RoboDK station: PaintingUV.rdk

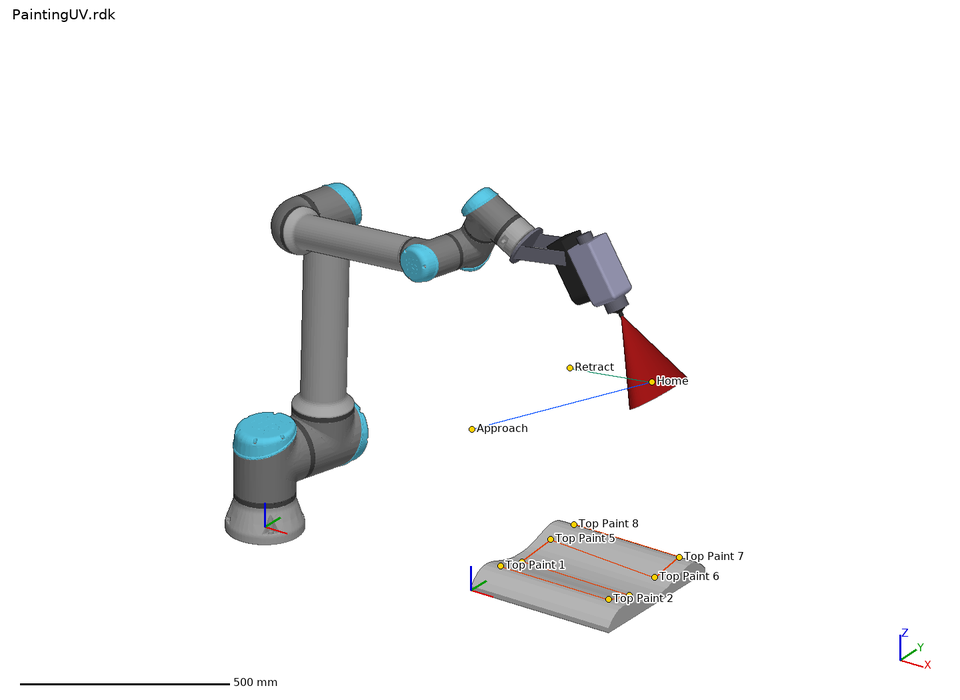
[picture v0: the station drawn from its stored meshes, robots at their saved joint values, targets as dots, program paths as lines]
Station PaintingUV (saved by RoboDK 5.9.0). Poses are relative to the parent item; angles as X-Y-Z fixed-axis rotations.
Station parameters (name, value as stored): LIN64
  - frame UR10e Base at (0, 0, 0) mm
    - robot UR10e: 6 axes, payload 10 kg, reach 1300 mm, repeatability 0.05 mm, weight 28.9 kg
        modified DH rows (alpha deg, a mm, theta deg, d mm): 0, 0, 0, 180.7; 90, 0, 180, 0; 0, 612.6, 0, 0; 0, 571.335, 0, 174.15; -90, 0, 0, 119.85; 90, 0, 180, 116.55
        joint limits [-360, -360, -360, -360, -360, -360] to [360, 360, 360, 360, 360, 360]; home [0, -90, -90, 0, 90, 0]; saved at [164.043, -88.205, 75.684, -137.69, -76.063, 82.15]
      - tool Paint gun, TCP at (50, 0, 450) mm, rotated rx 0 ry 30 rz 0 deg, size 203.2 x 279.7 x 471.5 mm
  - frame Frame 2 at (600, 0, 0) mm
    - object Object Inspection at (0, 0, 0) mm, size 400 x 400 x 46.2 mm, geometry from Object Inspection.stl
    - target Home (Cartesian target) at (532.05, -7.54, 703.9) mm, rotated rx -180 ry 31.17 rz 180 deg; joints [164.043, -88.205, 75.684, -137.69, -76.063, 82.15] of UR10e
    - target Approach (Cartesian target) at (7.39, -7.54, 431.89) mm, rotated rx 180 ry 0 rz 180 deg; joints [27.111, -58.336, -102.171, -82.294, 76.829, 113.912] of UR10e
    - target Retract (Cartesian target) at (7.39, 400, 431.89) mm, rotated rx 180 ry 0 rz -180 deg; joints [66.133, -75.4, -89.716, -91.735, 62.791, 152.938] of UR10e
    - target Top Paint 1 (Cartesian target) at (35, 72.72, 44.78) mm, rotated rx -168.77 ry 0.86 rz -179.92 deg; joints [48.293, -65.218, -137.407, -52.988, 60.349, 131.441] of UR10e
    - target Top Paint 2 (Cartesian target) at (350, 72.54, 44.95) mm, rotated rx -168.77 ry 0.86 rz -179.92 deg; joints [27.744, -99.255, -110.916, -35.769, 67.204, 109.799] of UR10e
    - target Top Paint 3 (Cartesian target) at (350, 157.15, 21.87) mm, rotated rx -164.84 ry -1.57 rz 179.79 deg; joints [34.896, -104.265, -105.486, -43.237, 62.641, 116.657] of UR10e
    - target Top Paint 4 (Cartesian target) at (35, 161.08, 21.16) mm, rotated rx -171.8 ry -0.46 rz 179.97 deg; joints [52.55, -70.997, -135.374, -50.46, 62.181, 137.077] of UR10e
    - target Top Paint 5 (Cartesian target) at (35, 281.13, 32.66) mm, rotated rx 162.41 ry -2.12 rz -179.67 deg; joints [40.418, -71.222, -139.459, -27.296, 84.151, 133.461] of UR10e
    - target Top Paint 6 (Cartesian target) at (350, 263.31, 27.46) mm, rotated rx 165.1 ry 1.52 rz 179.8 deg; joints [24.923, -101.47, -113.79, -20.179, 88.855, 118.594] of UR10e
    - target Top Paint 7 (Cartesian target) at (350, 365.32, 40.44) mm, rotated rx -154.99 ry -4.26 rz 179.06 deg; joints [48.617, -117.302, -83.383, -68.828, 55.066, 131.742] of UR10e
    - target Top Paint 8 (Cartesian target) at (35, 377.77, 33.39) mm, rotated rx -144.03 ry -8.69 rz 177.17 deg; joints [67.362, -107.854, -96.138, -90.311, 57.466, 154.888] of UR10e
  - program ApproachMove (4 instructions, listed below)
  - program PaintTop (10 instructions, listed below)
  - program RetractMove (4 instructions, listed below)
  - program MainProgram (11 instructions, listed below)
  - Python program SprayOn (listed below)
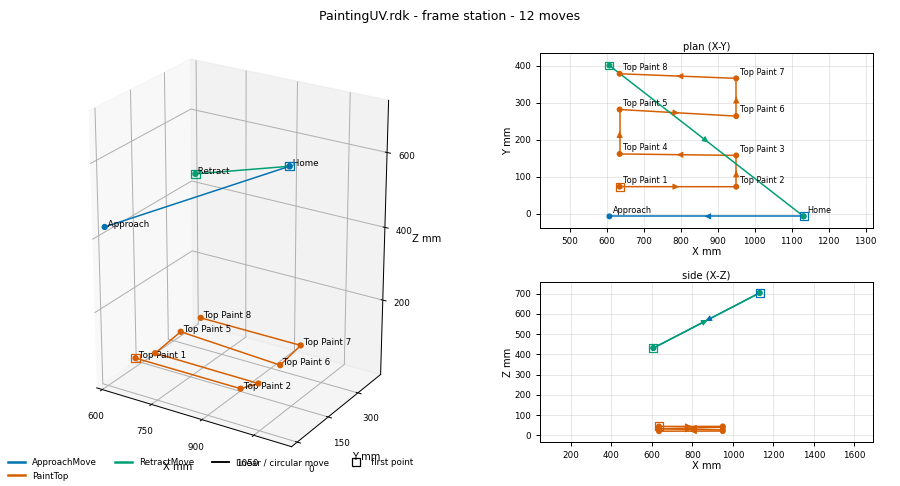
[picture p0: tool path of PaintingUV.rdk in frame station, 12 of 12 moves have a stored position in this frame; points joined in program order, loops and branches not executed]

--- program ApproachMove (robot UR10e) ---
  Set Ref.: Frame 2
  Set Tool: Paint gun
  MoveL (Home)
  MoveL (Approach)

--- program PaintTop (robot UR10e) ---
  Set Ref.: Frame 2
  Set Tool: Paint gun
  MoveL (Top Paint 1)
  MoveL (Top Paint 2)
  MoveL (Top Paint 3)
  MoveL (Top Paint 4)
  MoveL (Top Paint 5)
  MoveL (Top Paint 6)
  MoveL (Top Paint 7)
  MoveL (Top Paint 8)

--- program RetractMove (robot UR10e) ---
  Set Ref.: Frame 2
  Set Tool: Paint gun
  MoveL (Retract)
  MoveL (Home)

--- program MainProgram (robot UR10e) ---
  Call ApproachMove
  Call SprayOn(1)
  Call PaintTop
  Call SprayOn(1)
  Call PaintTop
  Call SprayOn(1)
  Call PaintTop
  Call SprayOn(1)
  Call PaintTop
  Call SprayOn(0)
  Call RetractMove

--- Python program SprayOn ---
# This macro allows simulating a spray gun for painting or to simulate the trace of inspaction
#
# You can call SprayOn(1) to simulate turning the Spray gun ON or SprayOn(0) to stop simulating the gun
# Calling SprayOn(-1) clears all displayed data
# The macro will output spray gun statistics
#
# --------------------------------------------------------------
# This script shows how to create "spray" object in RoboDK that allows simulating particle deposition by using:
# RDK.Spray_Add(tool, object, options_command, volume, geometry)
#    tool: tool item (TCP) to use
#    object: object to project the particles
#    options_command (optional): string to specify options.
#    volume (optional): Matrix of parameters defining the volume of the spray gun
#    geometry (optional): Matrix of vertices defining the triangles.
#
# More information here:
# https://robodk.com/doc/en/PythonAPI/robodk.html#robodk.robolink.Robolink.Spray_Add
# https://robodk.com/doc/en/RoboDK-API.html
#
# The scripts ArcStart, ArcEnd and WeldOn and SpindleOn behave in a similar way, the only difference is the default behavior
# This behavior simmulates Fanuc Arc Welding and triggers appropriate output when using the customized post processor.
# Select ESC to clear the trace manually.
#
# Example scripts that use Spray_Add:
#     SpindleOn / SpindleOff    -> Turn trace On/Off
#     ArcOn / ArcOff            -> Turn trace On/Off
#     SprayOn / SprayOff        -> Simulate a spray given a workspace volume (for painting)
#     WeldOn / WeldOff          -> Support for multiple weld guns

#------------------------------------------------------------------

# Use a specific tool as a spray gun
Tool_Name = None
#Tool_Name = 'Tool 2'

# Use a specific object to project particles:
Object_Name = None
#Object_Name = 'Part'

# Define the default action (0 to deactivate, +1 to activate, -1 to clear any spray gun simulation)
# Setting it to None will display a message
ACTION = None

from robodk.robolink import *  # API to communicate with RoboDK
from robodk.robomath import *  # basic matrix operations
from robodk.robodialogs import *

RDK = Robolink()

# quit if we are not in simulation mode
if RDK.RunMode() != RUNMODE_SIMULATE:
    quit()

# Get any previously added spray gun simulations and display statistics (spray on the part vs spray falling out of the part)
info, data = RDK.Spray_GetStats()
if data.size(1) > 0:
    print("Spray gun statistics:")
    print(info)
    print(data.tr())
    # # Diplay statistics
    # RDK.ShowMessage("Material used: %.1f%%<br>Material waisted: %.1f%%<br>Total particles: %.1f" % (data[1,0],data[2,0],data[3,0]), True)
    # # Clear previous spray
    # RDK.Spray_Clear()

# Check if we are running this program inside another program and passing arguments
import sys
if len(sys.argv) > 1:
    ACTION = int(sys.argv[1])

# If the default ACTION is None, display a message to activate/deactivate the spray gun
if ACTION is None:
    print('Note: This macro can be called as Spray(1) or SprayOn(0)')
    entry = mbox('Turn gun ON or OFF', ('On', '1'), ('Off', '0'))
    if not entry:
        quit()
    ACTION = int(entry)

if ACTION == 0:
    # Turn the gun off
    RDK.Spray_SetState(SPRAY_OFF)

elif ACTION < 0:
    # Clear all spray simulations (same as pressing ESC key)
    RDK.Spray_Clear()

elif ACTION > 0:
    # Create a new spray gun object in RoboDK
    # by using RDK.Spray_Add(tool, object, options_command, volume, geometry)
    # tool: tool item (TCP) to use
    # object: object to project the particles
    # options_command (optional): string to specify options. Example:
    #     STEP=AxB: Defines the grid to be projected 1x1 means only one line of particle projection (for example, for welding)
    #     PARTICLE: Defines the shape and size of particle (sphere or particle), unless a specific geometry is provided:
    #       a- SPHERE(radius, facets)
    #       b- SPHERE(radius, facets, scalex, scaley, scalez)
    #       b- CUBE(sizex, sizey, sizez)
    #     RAND=factor: Defines a random factor factor 0 means that the particles are not deposited randomly
    #     ELLYPSE: defines the volume as an ellypse (default)
    #     RECTANGLE: defines the volume as a rectangle
    #     PROJECT: project the particles to the surface (default) (for welding, painting or scanning)
    #     NO_PROJECT: does not project the particles to the surface (for example, for 3D printing)
    #
    # volume (optional): Matrix of parameters defining the volume of the spray gun
    # geometry (optional): Matrix of vertices defining the triangles.

    tool = 0  # auto detect active tool
    obj = 0  # auto detect object in active reference frame
    if Tool_Name is not None:
        tool = RDK.Item(Tool_Name, ITEM_TYPE_TOOL)

    if Object_Name is not None:
        obj = RDK.Item(Object_Name, ITEM_TYPE_OBJECT)
    # We can specify a given tool object and/or object
    #robot = RDK.Item("ABB IRB 2600-12/1.85", ITEM_TYPE_ROBOT)
    #tools = robot.Childs()
    #if len(tools) > 0:
    #    tool = tools[0]
    #obj = RDK.Item('object', ITEM_TYPE_OBJECT)

    options_command = "ELLYPSE PROJECT PARTICLE=SPHERE(4,8,1,1,0.5) STEP=8x8 RAND=2"  # simulate
    #options_command = "PARTICLE=CUBE(10,10,2) STEP=8x8"
    #options_command = "PARTICLE=SPHERE(4,8) STEP=8x8"
    #options_command = "PARTICLE=SPHERE(4,8,1,1,0.1) STEP=8x8 RAND=3"

    # Example commands for welding:
    # options_command = "PROJECT PARTICLE=SPHERE(4,8)"
    # options_command = PARTICLE=SPHERE(4,8) STEP=1x0

    # define the ellypse volume as p0, pA, pB, colorRGBA (close and far), in mm
    # coordinates must be provided with respect to the TCP
    close_p0 = [0, 0, -200]  # xyz in mm: Center of the conical ellypse (side 1)
    close_pA = [5, 0, -200]  # xyz in mm: First vertex of the conical ellypse (side 1)
    close_pB = [0, 10, -200]  # xyz in mm: Second vertex of the conical ellypse (side 1)
    close_color = [1, 0, 0, 1]  # RGBA (0-1)

    far_p0 = [0, 0, 50]  # xyz in mm: Center of the conical ellypse (side 2)
    far_pA = [60, 0, 50]  # xyz in mm: First vertex of the conical ellypse (side 2)
    far_pB = [0, 120, 50]  # xyz in mm: Second vertex of the conical ellypse (side 2)
    far_color = [0, 0, 1, 0.2]  # RGBA (0-1)

    close_param = close_p0 + close_pA + close_pB + close_color
    far_param = far_p0 + far_pA + far_pB + far_color
    volume = Mat([close_param, far_param]).tr()
    RDK.Spray_Add(tool, obj, options_command, volume)
    RDK.Spray_SetState(SPRAY_ON)

    # Another example with a varying rectancular shape
    # define the rectangular volume as p0, pA, pB, colorRGBA (close and far)
    # close_param = [-90,-117,  0,  90,-117,0,   -90,117,  0,       0.2,0.2,1,.1]
    # far_param   = [-175,-190,200, 175,-190,200,   -175,190,200,   0.5,0,0,.9]
    # volume = Mat([close_param, far_param])
    # RDK.Spray_Add(tool, obj, "RECTANGLE PARTICLE=SPHERE(2,5) STEP=15x15 RAND=3", volume.tr())
    # RDK.Spray_SetState(SPRAY_ON)

    # Optional: define geometry as a list of triangles with normals (instead of a scaled cube or a sphere)
    # geom = Mat([[0,0,0,   0,0,1], [5,0,0,   0,0,1], [0,5,0,   0,0,1]])
    # RDK.Spray_Add(tool, obj, "STEP=8x8 RANDX=3", volume.tr(), geom.tr())
    # RDK.Spray_SetState(SPRAY_ON)
